INTERFACE I_ForwardEnumerator extends I_Disposable

END_INTERFACE

(* stored: Version 1.1.0.1, ProductVersion 3.1.4024.12
   Itf I_ForwardEnumerator: Id {e9757b38-1996-45e6-a6c8-96fd1404a343} *)
